FUNCTION_BLOCK fileT_to_sysT
VAR_INPUT
	T_LoDW : DWORD;
	T_HiDW : DWORD;
END_VAR
VAR_OUTPUT
	sysT : TIMESTRUCT;
END_VAR
VAR
	fileT : T_FILETIME;
END_VAR

fileT.dwLowDateTime:= T_LoDW;			//change hex time to hh:mm:ss time
fileT.dwHighDateTime:= T_HiDW;
sysT := FILETIME_TO_SYSTEMTIME(fileT);

END_FUNCTION_BLOCK

(* stored: Version 1.1.0.1, ProductVersion 3.1.4024.3
   POU fileT_to_sysT: Id {49a9d259-4611-425a-8a32-dc2fbd4d2c02}, SpecialFunc None *)
